// TwinCAT 3 PLC project PLC_CocaCola_BottleFilling
// ProgramVersion: 3.1.4024.0
// libraries:
//   Tc2_Standard, * (Beckhoff Automation GmbH)
//   Tc2_System, * (Beckhoff Automation GmbH)
//   Tc3_Module, * (Beckhoff Automation GmbH)
// project tree:
//   / ConveyorTask_Cycle.TcTTO, ProductionTask_Cycle.TcTTO
//   GVLs/ GVL_CocaCola.TcGVL (not stored)
//   POUs/ CalculateFillTimeTask.TcPOU, ConveyorTask.TcPOU, ProductionTask.TcPOU (not stored)
// real-time tasks:
//   TASK PlcTask: cycle T#10ms, priority 20, ADS port 350
//   TASK ConveyorTask_Cycle: cycle T#10ms, priority 22, ADS port 350
//   TASK ProductionTask_Cycle: cycle T#50000us, priority 23, ADS port 351

CONFIGURATION PLC_CocaCola_BottleFilling
    RESOURCE PLC ON TwinCAT3
        TASK ConveyorTask_Cycle(INTERVAL := T#10ms, PRIORITY := 22);
        TASK ProductionTask_Cycle(INTERVAL := T#50000us, PRIORITY := 23);
        PROGRAM ConveyorTask WITH ConveyorTask_Cycle : ConveyorTask;
        PROGRAM ProductionTask WITH ProductionTask_Cycle : ProductionTask;
    END_RESOURCE
END_CONFIGURATION

// ---- POUs/ConveyorTask.TcPOU
PROGRAM ConveyorTask
VAR
  DebounceTON : TON;   // Debounce timer for bottle detection
  EvacuateTON : TON;    // Timer for moving the filled bottle away
  State : INT := 0;    // 0 = RUNNING, 1 = STOPPED, 2 = EVACUATE
END_VAR


CASE State OF

  // The idea proposed divides the 3 actions the conveyor belt will do, run, stop and evacuate if error found
	
  // State 0 → RUNNING (conveyor moving and waiting)
	
 0:
  gConveyorStateStr := 'RUNNING';
  gActuator_ConveyorRun := TRUE;

   // Debounce the bottle sensor gives stability, so when sensor reaches 100MS it will -> go into true
   DebounceTON(IN := gSensor_BottleDetected, PT := T#100MS);

   // When the bottle is detected firmly → stop conveyor, if it detects the bottle then its stops moving
    IF DebounceTON.Q THEN
     gActuator_ConveyorRun := FALSE;
     gBottleReadyForFill := TRUE;    // here we tell ProductionTask to start filling, connecting both procedures
     gConveyorStateStr := 'STOPPED';	// Visual represnetation that the conveyor has stopped
     State := 1;		// Go to Stop
      END_IF


    // State 1 → STOPPED (waiting for filling to complete) 
	
	
    1:
       gConveyorStateStr := 'STOPPED';
       gActuator_ConveyorRun := FALSE; // Running stopped waiting for bottle to be completly full

       // When ProductionTask communicates the bottle is already full
       IF gBottleFilled THEN
       gBottleReadyForFill := FALSE;
        EvacuateTON(IN := FALSE);      // reset timer
        State := 2;                  // go to EVACUATE
        END_IF



	// STATE 2 → EVACUATE (push filled bottle away)

	2:
		gConveyorStateStr := 'EVACUATE';
		gActuator_ConveyorRun := TRUE; // When bottle is full we want the conveyor to reactivate so it pushes away the filled bottle

		EvacuateTON(IN := TRUE, PT := T#800MS); // This is to give some margin of evacuation

		IF (NOT gSensor_BottleDetected) AND EvacuateTON.Q THEN // If there is no bottle + the timer ends
		gBottleFilled := FALSE;
		EvacuateTON(IN := FALSE);
		 State := 0;				// We go back to running   
		 END_IF

END_CASE

END_PROGRAM

// ---- POUs/CalculateFillTimeTask.TcPOU
FUNCTION CalculateFillTime_ms : DINT
VAR_INPUT
    vol_l   : REAL;   // Bottle volume [L]
    rate_Ls : REAL;   // Fill rate [L/s]
END_VAR
VAR
    t_ms : REAL;      // Calculated time in milliseconds
END_VAR



// Basic validation (avoid division by zero)
IF rate_Ls <= 0 THEN
    CalculateFillTime_ms := 0;
    RETURN;
END_IF

// Convert time from seconds to milliseconds
t_ms := (vol_l / rate_Ls) * 1000.0;

// Clamp limits (just to avoid impossible values)
IF t_ms < 0.0 THEN
    t_ms := 0.0;
ELSIF t_ms > 60000.0 THEN
    t_ms := 60000.0;   // 60 seconds max
END_IF

// Return the calculated time as DINT
CalculateFillTime_ms := REAL_TO_DINT(t_ms);

END_FUNCTION
